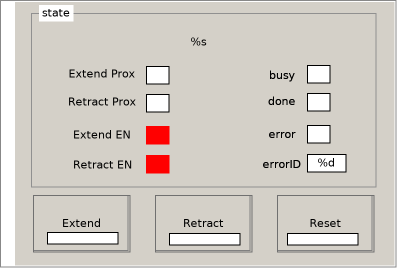
VISUALIZATION Cylinder  // 397x268
VAR_IN_OUT
	userdata : Cylinder_HMI_Structure;
END_VAR
    Rectangle (14,1 381x265)
    GroupBox (31,5 345x182), "state"
        Rectangle (276,60 23x18), colour toggle: userData.busy
        Rectangle (276,88 23x18), colour toggle: userData.done
        Rectangle (276,120 23x18), colour toggle: userData.error
        Rectangle (276,149 39x18), "%d", text variable: userData.errorID, colour toggle: userData.errorID
        Rectangle (115,61 23x18), colour toggle: userData.bExtend_Prox
        Rectangle (115,89 23x18), colour toggle: userData.bRetract_Prox
        Rectangle (115,121 23x18), colour toggle: userData.bExtend_Enable
        Label (191,52 120x37), "busy"
        Label (191,78 120x37), "done"
        Label (191,111 120x37), "error"
        Label (191,141 120x37), "errorID"
        Rectangle (115,150 22x18), colour toggle: userData.bRetract_Enable
    Rectangle (62,27 273x30), "%s", text variable: userData.errorTXT, colour toggle: userData.errorTXT
    Rectangle (307,65 23x18), colour toggle: userData.busy
    Rectangle (307,93 23x18), colour toggle: userData.done
    Rectangle (307,125 23x18), colour toggle: userData.error
    Rectangle (307,154 39x18), "%d", text variable: userData.errorID, colour toggle: userData.errorID
    Rectangle (146,66 23x18), colour toggle: userData.bExtend_Prox
    Rectangle (146,94 23x18), colour toggle: userData.bRetract_Prox
    Rectangle (146,126 23x18), colour toggle: userData.bExtend_Enable
    Label (222,57 120x37), "busy"
    Label (222,83 120x37), "done"
    Label (222,116 120x37), "error"
    Label (222,146 120x37), "errorID"
    Rectangle (146,155 23x18), colour toggle: userData.bRetract_Enable
    Group (33,195 97x57)
        Button (0,0 97x57), "Extend"
            tap userData.bExtend_jog
        Rectangle (14,37 71x12), colour toggle: userData.bExtend_Work
    Group (155,195 97x57)
        Button (0,0 97x57), "Retract"
            tap userData.bRetract_jog
        Rectangle (14,38 71x12), colour toggle: userData.bRetract_Work
    Group (277,195 97x57)
        Button (0,0 97x57), "Reset"
            tap userData.bReset_Error
        Rectangle (10,38 71x12), colour toggle: userData.error
    Group (27,59 150x121)
        Label (0,0 150x30), "Extend Prox"
        Label (0,28 150x30), "Retract Prox"
        Label (0,61 150x30), "Extend EN"
        Label (1,91 149x30), "Retract EN"
END_VISUALIZATION

(* stored: Version 1.1.0.1, ProductVersion 3.1.4018.5
   Visu Cylinder: Id {48544263-0481-41e1-91e2-7f8e008d7f22} *)
